{attribute 'qualified_only'}
{attribute 'strict'}
TYPE E_Beckhoff_EL6001_State :
(
	INIT,
	READY,
	TRANSMIT, 
	RECEIVE
);
END_TYPE

(* stored: Version 1.1.0.1, ProductVersion 3.1.4024.12
   DUT E_Beckhoff_EL6001_State: Id {88379d5f-ba1e-00fd-19ab-2fc9c8b737cb} *)
